(* LS Electric XG5000 project: Dol_Starter *)
(* PLC LSPLC *)

PROGRAM NewProgram (* task: Scan Program *)
VAR
    Motor AT %QX0.0.0 : BOOL;
    Start AT %IX0.0.0 : BOOL;
    Stop AT %IX0.0.1 : BOOL;
END_VAR

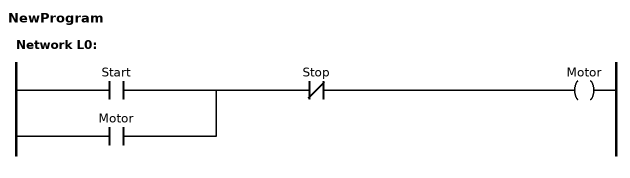
(* Rung L0 *)
Motor := (Start OR Motor) AND NOT Stop;
END_PROGRAM